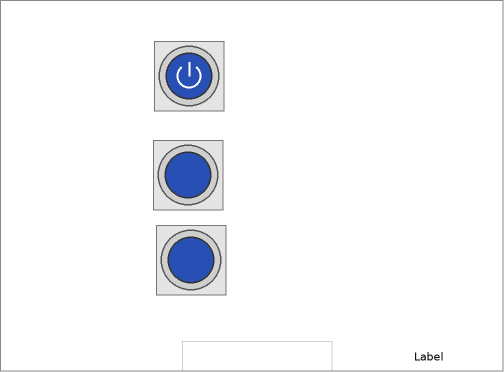
VISUALIZATION HMI  // 504x372
    PushSwitch (153,140 70x70), behaviour: TOGGLE, style: Switch-PushSwitch-Blue
    PowerSwitch (154,41 70x70), behaviour: TOGGLE, style: Switch-PowerSwitch-Blue
    PushSwitchLed (156,225 70x70), behaviour: TOGGLE, style: Switch-PushSwitchLed-Blue
    Textfield (182,341 150x30)
    Label (354,342 150x30), "Label"
END_VISUALIZATION

(* stored: Version 1.1.0.1, ProductVersion 3.1.4024.11
   Visu HMI: Id {e83fe0f6-a3fa-41e5-916a-5fed390733ae} *)
